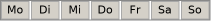
VISUALIZATION V_WeekDay  // 211x21
VAR_IN_OUT
	eWeekDay : E_WeekDay;
END_VAR
    Rectangle (1,1 28x18), "Mo", colour toggle: eWeekDay = 1
        OnMouseUp: execute { eWeekDay := 1; }
    Rectangle (31,1 28x18), "Di", colour toggle: eWeekDay = 2
        OnMouseUp: execute { eWeekDay := 2; }
    Rectangle (61,1 28x18), "Mi", colour toggle: eWeekDay = 3
        OnMouseUp: execute { eWeekDay := 3; }
    Rectangle (91,1 28x18), "Do", colour toggle: eWeekDay = 4
        OnMouseUp: execute { eWeekDay := 4; }
    Rectangle (121,1 28x18), "Fr", colour toggle: eWeekDay = 5
        OnMouseUp: execute { eWeekDay := 5; }
    Rectangle (151,1 28x18), "Sa", colour toggle: eWeekDay = 6
        OnMouseUp: execute { eWeekDay := 6; }
    Rectangle (181,1 28x18), "So", colour toggle: eWeekDay = 0
        OnMouseUp: execute { eWeekDay := 0; }
END_VISUALIZATION

(* stored: Version 1.1.0.1, ProductVersion 3.1.4018.9
   Visu V_WeekDay: Id {b0cb990e-efcd-445b-82d2-537f29c1a9e0} *)
